PROGRAM POU_Test
VAR
	fbSimpleLinearTwoWayDriveTest: FB_SimpleLinearTwoWayDrive_Test; 
	fbLinearMovementWithFeedbackTest: FB_LinearMovementWithFeedbackTest;
	fbSewMovitracBFieldbusTest: FB_SewMovitracBFieldbusTest;
END_VAR

TcUnit.RUN();

END_PROGRAM

(* stored: Version 1.1.0.1, ProductVersion 3.1.4024.11
   POU POU_Test: Id {196e0b9a-9deb-4dd0-a48f-8902bcc60beb}, SpecialFunc None *)
